FUNCTION_BLOCK FB_DoubleContactor EXTENDS FB_Contactor IMPLEMENTS I_DriveDouble
VAR
	_outputReverse	AT%Q* : BOOL;	// Switch variable to start/stop Reverse psychical output
END_VAR

{warning 'add method implementation '}
METHOD SwitchReverseOff : BOOL
_outputReverse := False;
END_METHOD

{warning 'add method implementation '}
METHOD SwitchReverseOn : BOOL
_outputReverse := True;
END_METHOD

END_FUNCTION_BLOCK

(* stored: Version 1.1.0.1, ProductVersion 3.1.4024.12
   POU FB_DoubleContactor: Id {cc7fc58b-d311-4e65-ad7d-7841037b2b38}, SpecialFunc None
   Method SwitchReverseOff: Id {5505444f-14b2-4f81-9446-45e904c6b051}
   Method SwitchReverseOn: Id {383937bc-a274-4aa8-97cc-b7751262242e} *)
